// TIA Portal V20 export
DATA_BLOCK "DB_OPC_RealTime"   // DB104
{ S7_Optimized_Access := 'TRUE' }
// stored: MemoryReserve 100
   VAR
      GripperUndrilledClampOpen : Bool;   // Test
      GripperUndrilledClampClosed : Bool;   // Test
      FixturePosition : Real;   // Test
      X_AxisBrakePressCtrl : Bool;   // Digital Input
      Y_AxisBrakePressCtrl : Bool;   // Digital Input
      BreakerCtrl : Bool;   // Digital Input
      CabinetTemperatureCtrl : Bool;   // Digital Input
      UpsPowerFailure : Bool;   // Digital Input
      AirPressureCtrl : Bool;   // Digital Input
      ShutterClosed : Bool;   // Digital Input
      AirDryerOK : Bool;   // Digital Input
      UPS_BatteryOK : Bool;   // Digital Input
      FrontDoorClosed : Bool;   // Digital Input
      InfeedReadyOkStart : Bool;   // Digital Input
      CoolingOK : Bool;   // Digital Input
      PowerReady : Bool;   // Digital Input
      AlarmI2T : Bool;   // Digital Input
      HeadLaserBusy : Bool;   // Digital Input
      HeadLaserBreaker : Bool;   // Digital Input
      FrontDoorLocked : Bool;   // Digital Input
      UPS_CommonAlarm : Bool;   // Digital Input
      UPS_BatteryLow : Bool;   // Digital Input
      HeadChillerHighPressure : Bool;   // Digital Input
      HeadChillerWaterTemperature : Bool;   // Digital Input
      HeadChillerFlow : Bool;   // Digital Input
      HeadChillerCollectivFault : Bool;   // Digital Input
      HeadChillerWaterLevel : Bool;   // Digital Input
      UpsByPassActive : Bool;   // Digital Input
      HeadChillerAmbiantTemperature : Bool;   // Digital Input
      LoadClampOpened : Bool;   // Digital Input
      LoadClampNotClosedWithPart : Bool;   // Digital Input
      UnloadClampOpened : Bool;   // Digital Input
      UpsFault : Bool;   // Digital Input
      InternalGateLocked : Bool;   // Digital Input
      ExternalGateLocked : Bool;   // Digital Input
      InverterActive : Bool;   // Digital Input
      UnloadClampNotClosedWithPart : Bool;   // Digital Input
      InternalGateOpened : Bool;   // Digital Input
      ExternalGateOpened : Bool;   // Digital Input
      PowerMeterBackCtrl : Bool;   // Digital Input
      PowerMeterFrontCtrl : Bool;   // Digital Input
      HeadChillerCutOff : Bool;   // Digital Input
      HeadChillerTemperature : Bool;   // Digital Input
      ClampingOpenCtrl : Bool;   // Digital Input
      B_AxisBrakeReleasedCtrl : Bool;   // Digital Input
      B_AxisReferencePoint : Bool;   // Digital Input
      SourceChillerHighPressure : Bool;   // Digital Input
      SourceChillerWaterTemperature : Bool;   // Digital Input
      SourceChillerFlow : Bool;   // Digital Input
      SourceChillerCollectivFault : Bool;   // Digital Input
      SourceChillerWaterLevel : Bool;   // Digital Input
      SourceChillerAmbiantTemperature : Bool;   // Digital Input
      SourceChillerCutOff : Bool;   // Digital Input
      SourceChillerTemperature : Bool;   // Digital Input
      OperatingCounter : Bool;   // Digital Output
      GeneralAirValve : Bool;   // Digital Output
      SmartLineDisable : Bool;   // Digital Output
      MachineLight : Bool;   // Digital Output
      MachineLightBack : Bool;   // Digital Output
      LightTowerOrange : Bool;   // Digital Output
      LightTowerRed : Bool;   // Digital Output
      LightTowerBlue : Bool;   // Digital Output
      LightTowerGreen : Bool;   // Digital Output
      LightTowerWhite : Bool;   // Digital Output
      Backlight : Bool;   // Digital Output
      InfeedON : Bool;   // Digital Output
      AxisActivation : Bool;   // Digital Output
      BuzzerActivation : Bool;   // Digital Output
      ElbaronPowerON : Bool;   // Digital Output
      ObservationCameraLight : Bool;   // Digital Output
      LaserExternalDoorOpening : Bool;   // Digital Output
      CoolingStart : Bool;   // Digital Output
      X_AxisBrakeActivation : Bool;   // Digital Output
      Y_AxisBrakeActivation : Bool;   // Digital Output
      AxisB_TeachInClampingPart : Bool;   // Digital Output
      EPO_UPS : Bool;   // Digital Output
      HeadLaserStart : Bool;   // Digital Output
      HeadLaserStop : Bool;   // Digital Output
      Axis2_PowerContactor : Bool;   // Digital Output
      GasAssistOn : Bool;   // Digital Output
      SmartLineReset : Bool;   // Digital Output
      XY_AxisPowerContactor : Bool;   // Digital Output
      LaserAirPressureProcess : Bool;   // Digital Output
      Bus60V_PowerContactor : Bool;   // Digital Output
      LoadClampClosing : Bool;   // Digital Output
      LoadClampOpening : Bool;   // Digital Output
      UnloadClampClosing : Bool;   // Digital Output
      UnloadClampOpening : Bool;   // Digital Output
      ClampingOpening : Bool;   // Digital Output
      ClampingClosing : Bool;   // Digital Output
      B_AxisBrakeRelease : Bool;   // Digital Output
      Suction : Bool;   // Digital Output
      ExternalGateClosing : Bool;   // Digital Output
      ExternalGateOpening : Bool;   // Digital Output
      InternalGateClosing : Bool;   // Digital Output
      InternalGateOpening : Bool;   // Digital Output
      PowerMeterRetract : Bool;   // Digital Output
      PowerMeterAdvance : Bool;   // Digital Output
      Blowing : Bool;   // Digital Output
      LaserPowerMeter : Real;   // Analog Input
      AxisB_ClampingPart : Real;   // Analog Input
      LaserAirPressureProcess_1 : Real;   // Analog Input
      InletAirPressure : Real;   // Analog Input
      AmbiantTemperature : Real;   // Analog Input
      MachineTemperature : Real;   // Analog Input
      Cold_WaterTemperatureInput { ExternalWritable := 'False'} : Real;   // Analog Input
      Cold_WaterTemperatureOutput : Real;   // Analog Input
      X_AxisTemperaturePT1000 : Real;   // Analog Input
      Y_AxisTemperaturePT1000 : Real;   // Analog Input
      X_AxisTemperaturePTC : Real;   // Analog Input
      Y_AxisTemperaturePTC : Real;   // Analog Input
      NozzleOverpressure : Real;   // Analog Input
      OpticalPathOverpressure : Real;   // Analog Input
      LaserHeadOverpressure : Real;   // Analog Input
      ZLAxisOverpressure : Real;   // Analog Input
      XYAxisOverpressure : Real;   // Analog Input
      LeftAspiration : Real;   // Analog Input
      RightAspiration : Real;   // Analog Input
      ClimTemperature : Real;   // Analog Input
      SensorControllerStation1 : Real;   // Analog Input
      CabinetTemperature : Real;   // Analog Input
      NozzleOverpressureSetPoint : Real;   // Analog Output
      VentilatorSetPoint : Real;   // Analog Output
      PropValveClimSetPoint : Real;   // Analog Output
   END_VAR
BEGIN
END_DATA_BLOCK
